Fanuc KAREL source: KO00114.KL

PROGRAM KO00114
%NOLOCKGROUP
VAR
  A: ARRAY[2] OF BYTE
  B: INTEGER
  OUT: REAL
BEGIN
  A[1] = 1
  B = 2
  OUT = ATAN2(A[1], B)
END KO00114
